TYPE ST_ProcessCycleStatus :
STRUCT
    // GENERAL
    eState                         : E_CycleState;
    eMessage                       : E_ProcessCycleMessage;
    bActive                        : BOOL;
    bIdle                          : BOOL;
    bCompletePulse                 : BOOL;
    bFaulted                       : BOOL;
	bTimeoutFault        		   : BOOL;

    // WAIT CONDITIONS
    bWaitingForPart                : BOOL;
    bWaitingForOperator            : BOOL;
    bWaitingForIndex               : BOOL;
    bWaitingForSupports            : BOOL;

    // SUPPORTS
    bSiliconeSupportExtended       : BOOL;
    bSiliconeSupportRetracted      : BOOL;
    bAssemblySupportExtended       : BOOL;
    bAssemblySupportRetracted      : BOOL;

    // PROCESS SIMULATION
    bSiliconeProcessRunning        : BOOL;
    bSiliconeProcessComplete       : BOOL;
    bAssemblyProcessRunning        : BOOL;
    bAssemblyProcessComplete       : BOOL;

    // MESSAGE
    sMessage                       : STRING(255);
	
END_STRUCT
END_TYPE

(* stored: Version 1.1.0.1, ProductVersion 3.1.4026.18
   DUT ST_ProcessCycleStatus: Id {2e2ea3aa-1e0a-4f05-a304-4b64a12f3e81} *)
